(* CODESYS project Structs.export

Project tree, tasks and I/O mapping:
  Structs/
    data type BitByte
    data type udtActuator
    data type udtCamera
    data type udtGeneralBuffer
    data type udtGornModbus
    data type udtTMPBreakingValve
    data type udtVacuumCamera
    DiscreteSignal/
      data type udtDiscreteSignal
      data type udtDiscreteSignalSetting
    Driver/
      data type udtBSDDriver
      data type udtBSDDriverSetting
    FVP/
      data type udtFVP
      data type udtFVPSetting
    GasRegulator/
      data type udtPIDSetting
    Gorn/
      data type udtGorn
      data type udtGornSetting
      Modbus/
        data type GornReadRegister
        data type GornWriteRegister
    HeatfloatSencore/
      data type udtHeatFloatSensore
      data type udtHeatFloatSensoreSetting
    Inficon/
      data type udtInficonGeneralCommand
      data type udtInficonGeneralParameters
      data type udtInficonMaterialParameters
      data type udtInficonProcessMaterialParameters
      data type udtInficonRemoteGeneral
      data type udtInficonRemoteMaterial
      data type udtInficonSensorParameter
      data type udtInficonSourceParameters
      data type udtInficonStatusGeneral
      data type udtInficonStatusMaterial
      data type udtInficonStatusSensor
      InficonType/
        data type InficonFloat
        data type InficonInteger
        data type InficonLong
        data type InficonTime
        BitByte/
          data type InficonInputStatus
          data type InficonLogicstatementStatus
          data type InficonOutputStatus
        Real/
          data type REAL3x1
          data type REAL41
          data type REAL4F31
          data type REAL4x2
          data type REAL5F32
          data type REAL5x3
          data type REAL6F32
    IPS/
      data type udtIPS
      data type udtIPSModbus
      Modbus/
        data type IpsMagnetronReadRegisters
        data type IpsMagnetronWriteRegisters
    Modbus/
      data type sModbusRegister
      data type unRegisterValue
    OWEN/
      data type OwenValue
    OwenAnalogSignal/
      data type udtOwenAnalogSignal
    Pumping/
      VacuumProccessWithSHV/
        data type udtVacuumProccessStatusBitMap
        data type udtVacuumProcess
        data type udtVacuumProcessState
        data type VacuumProccessStatus
        data type VacuumStage
        Devacuum/
          data type DevacuumUnitStage
          data type udtDevacuumUnitProcessSetting
        Revacuum/
          data type RevacuumStage
          data type udtRevacuumProcessSetting
        StartUnitStage/
          data type StartUnitStage
          data type udtStartUnitProcessSetting
        StopUnit/
          data type StopUnitStage
    RRG/
      data type udtRRG
      data type udtRRGSetting
      Modbus/
        data type udtRRGFlagState1
        data type udtRRGFlagState1Flags
        data type udtRRGFlagState2
        data type udtRRGFlagState2Flags
        data type udtRRGModbus
    Shutter/
      data type udtShutter
    TMPDigital/
      data type udtTMPDigital
      data type udtTMPDigitalSetting
    TRM151_Control/
      data type udtTRMHeaterView
      View/
        data type udtTRMChannelView
        data type udtTRMInputView
        data type udtTRMOutput
        Operating/
          data type udtTRMOperatingView
        Regulator/
          data type udtTRMPIDRegualtor
          data type udtTRMRegulatorView
        SetPoints/
          data type udtStepSetPointView
        TechnologProgramm/
          data type udtTRMTechnologOperation
          data type udtTRMTechnologOperationProgram
          data type udtTRMTechnologOperationProgramStep
    TRM151_Protocol/
      data type udtChannel
      data type udtTRM151_01
      Calculator/
        data type udtCalculator
        data type udtCalculatorInput
        data type udtCalculators
      Inputs/
        data type udtInput
        data type udtInputs
      LockAndChangeMode/
        data type udtTRMLockAndChangeMode
      OperationParameters/
        data type udtOperationParameters
        data type udtPowerFeedback
        data type udtSetPointFeedback
      Program/
        data type udtProgram
        data type udtProgramOfTechnolog
        data type udtStep
      Regulators/
        data type udt2PositionRegulator
        data type udtPIDRegulator
        data type udtRegulator
        data type udtRegulators
      SetPoint/
        data type udtProgramSetPoint
        data type udtSetPoints
        data type udtStepSetPoint
      SignalConverter/
        data type udtSignalConverter
        data type udtSignalConverters
    VacuumSensore/
      data type udtAPG100
      data type udtAPG100Setting
      data type udtPressureSensore
      data type udtPressureSensoreSettiing
    Valve/
      data type udtValve
      data type udtValveSetting
*)

// Structs/BitByte
TYPE BitByte :
STRUCT
	b0: BIT;
	b1: BIT;
	b2: BIT;
	b3: BIT;
	b4: BIT;
	b5: BIT;
	b6: BIT;
	b7: BIT;
END_STRUCT
END_TYPE

// Structs/udtActuator
TYPE udtActuator :
	(*Стурктура для Актуатора*)
STRUCT
	xInterlock:				BOOL;// INPUT: Внешняя блокировка
	xOpenInterlock:			BOOL;
	xCloseInterlock:		BOOL;
	xOpenBlocked:			BOOL;
	xCloseBlocked:			BOOL;
	xServiceMode:			BOOL;// COMMAND: Сервисный режим
	xOpenCommand:			BOOL;// COMMAND: Команда на октрытие
	xCloseCommand:			BOOL;// COMMAND: Команда на закрытие
	xOpen:					BOOL;// OUTPUT: Открытие
	xClose:					BOOL;// OUTPUT: Закрытие
END_STRUCT
END_TYPE

// Structs/udtCamera
TYPE udtCamera :
	(*Структура для обработки состояния камеры*)
STRUCT
	xOpened:				BOOL;//INPUT: Камера открыта
	xClosed:				BOOL;//INPUT: Камера закрыта
	xUpPosition:			BOOL;//INPUT: Верхняя позиция
END_STRUCT
END_TYPE

// Structs/udtGeneralBuffer
TYPE udtGeneralBuffer :
STRUCT
	Buffer: POINTER TO BYTE;
	MaxLength: INT;
	Offset: INT;
END_STRUCT
END_TYPE

// Structs/udtGornModbus
TYPE udtGornModbus :
STRUCT
	uiModbusAddress: UINT;//Адрес юнита
	Read:			GornReadRegister;//Список всех регистров на чтение
	Write:			GornWriteRegister;//Список всех регистров на запись
	
END_STRUCT
END_TYPE

// Structs/udtTMPBreakingValve
TYPE udtTMPBreakingValve :
STRUCT
	xAutoMode:			BOOL;//manual/Auto Mode
	xInterlock:			BOOL;
	xManualCommand: 	BOOL;
	xAutoCommand:		BOOL;
	xClosed:			BOOL;
	xOutputCommnad:		BOOL;
END_STRUCT
END_TYPE

// Structs/udtVacuumCamera
(*Структура данных для вакуумнйо камеры*)
TYPE udtVacuumCamera :
STRUCT
	xClosed:								BOOL;	//STATE: Вакуумная камер Открыта/Закрыта
	xCameraIsVaccumed: 						BOOL;	//STATE: Вакуумная система Остановлена/Запущена
	xFVPChecked:							BOOL;	//STATE: Форвакуумный насос прошел проверку
	VacuumCameraProcessStage:				INT;	//STATE: Стадия процесса вакуумной камеры
	
	
	
	rTmpForvacuumingProcessDonePressuresSp: REAL;	//Давление необходимое и достаточное для включения ТМН
	rPressureForVacuumiongProcessComplete:  REAL;	//давление для завершения процесса откачки
	tStopTMPtime:							TIME;  	//Полное время для остановки ТМН
	tOpenBAV3time:							TIME;   //период во времени при полной остановке ТМН когда будет открыьт клапан напуска
	
END_STRUCT
END_TYPE

// Structs/DiscreteSignal/udtDiscreteSignal
TYPE udtDiscreteSignal :
STRUCT
	xSignal:			BOOL;// I/O 

	xValue:				BOOL;// Ready value from/to PLC programms	
END_STRUCT
END_TYPE

// Structs/DiscreteSignal/udtDiscreteSignalSetting
TYPE udtDiscreteSignalSetting :
STRUCT
	xInv:				BOOL;// Инвертирвоанный сигнал
	xSimMode:			BOOL;// Simulation Mode
	xSimValue:			BOOL;// Simulation Value
END_STRUCT
END_TYPE

// Structs/Driver/udtBSDDriver
TYPE udtBSDDriver :
STRUCT
	AutoMode: 			BOOL;	//STATUS
	ServiceMode:		BOOL;	//STATUS
	Blocked:			BOOL;	//STATUS
	Run:				BOOL;	//STATUS
	
	
	
	rSpeedSP:			REAL;	//Setpoint
	
	xAutoCommand:		BOOL;	//COMMAND
	xManualCommand:		BOOL;	//COMMAND
	
	xInterlockSignal: 	BOOL; //Input
	xAlarmSignal:		BOOL; //Input
	
	xStartSignal:		BOOL;
	xCCWSignal:			BOOL;
	rSignal: 			REAL; //OUTPUT: CommandSignal to BSD driver Limit 0-5V
END_STRUCT
END_TYPE

// Structs/Driver/udtBSDDriverSetting
TYPE udtBSDDriverSetting :
STRUCT
	rMinSignalLimit:	REAL;
	rMaxSignalLimit:	REAL;
	rManualSpeedSP:		REAL;
	rAutoSpeedSP:		REAL;
	rMaxSpeed:			INT; //Оборы в минкуту
	xAutoMode:			BOOL;
	xServiceMode:		BOOL;
	xCCWMode:			BOOL;		
END_STRUCT
END_TYPE

// Structs/FVP/udtFVP
TYPE udtFVP :
	(*Структура данных форвакуумного насоса*)
STRUCT
	xPowerOnFeedBack:			BOOL;// INPUT: Обратная связь по питанию
	xInterlock:					BOOL;// INPUT: Внешний сигнал о блокировки
	xManualCommand:				BOOL;// COMMAND: Ручная комманда
	xAutoCommand:				BOOL;// COMMAND: Команда в автоматическом режиме
	xTurnOn:					BOOL;//	STATUS: Насос включен
	xBlocked:					BOOL;// OUTPUT: Сигнал о блокировке 
	xStart:						BOOL;// OUTPUT: Старт/Стоп ФВН
	xPowerOn:					BOOL;// OUTPUT: Состояние питания
END_STRUCT
END_TYPE

// Structs/FVP/udtFVPSetting
TYPE udtFVPSetting :
STRUCT
	xAutoMode:					BOOL;// COMMAND: Автоматическийй/ручной режим
	xServiceMode:				BOOL;// COMMAND: Сервисный режим
	
	xWithOutTurnOn:				BOOL;//Setting: Работа без контактора
END_STRUCT
END_TYPE

// Structs/GasRegulator/udtPIDSetting
TYPE udtPIDSetting :
STRUCT
	rMaunalSP: 	REAL; 	// Расход в литрах РРГ
	rAutoSP:	REAL;	// Необходимое давление.
	rMaxSP:		REAL; 	// Максимальный расход
	rMinSP:		REAL; 	// Минмиальный расход
	iP:			REAL; 	// Пропорциональынй коэффтициент
	tI:			REAL;	// Интегральный коэфф
	rK1RRG:		REAL;	// Коэффитциент РРГ
	rK2RRG:		REAL;
	rK3RRG:		REAL;
	
	xAutoMode:	BOOL;
END_STRUCT
END_TYPE

// Structs/Gorn/udtGorn
TYPE udtGorn :
	(*Стурктура данных для высокотемпературного нагревателя ГОРН
		Верхний уровень управления*)
STRUCT
	
	rSpCurrentFeedback:			REAL;// FEEDBACK: Обратная связь по уставке силы тока
	rSpVoltageFeedback:			REAL;// FEEDBACK: Обратная связь по уставке напряжения
	rFbCurrent:					REAL;// FEEDBACK: Обратная связь по силе тока
	rFbVoltage:					REAL;// FEEDBACK: Обратная связь по напряжению 
	xPowerOnFeedback:			BOOL;// INPUT: Обратная связь по питанию
	xInterlock:					BOOL;// INPUT: Внешняя блокировка
	xRemote:					BOOL;// COMMAND: местынй/дистанционный режимы работы
	xAutoMode:					BOOL;// COMMAND: ручной/автоматический режимы
	xManualCommand:				BOOL;// COMMAND: Команда выкл/вкл в ручном режиме
	xManualPowerCommand:		BOOL;// COMMAND: Команда выкл/вкл питания силовой части в ручном режиме.
	xAutoCommand:				BOOL;// COMMAND: Команда в автоматическом режиме
	xAutoPowerCommand:			BOOL;// COMMAND: Команда питания силовой части в автоматичсеском режиме
	xAcknowledge:				BOOL;// COMMAND: Оператор сбрасывает ошибки
	xBlocked:					BOOL;// STATUS: Заблокирован
	xTurnOn:					BOOL;//	STATUS: В работе
	xError:						BOOL;// STATUS: Общие ошибки
	xInternalError:				BOOL;// OUTPUT: Внутренняя ошибка
	xStabVoltageError:			BOOL;// OUTPUT: Ошибка стабилизации напряжения
	xStabCurrentError:			BOOL;// OUTPUT:	Ошибка стабилизации силы тока
	xPowerError:				BOOL;// OUTPUT: Ошибка силовой части
	xHeatProtect:				BOOL;// OUTPUT: Тепловая защита
	xRemoteStatus:				BOOL;// OUTPUT: Статус удаленной работы
END_STRUCT
END_TYPE

// Structs/Gorn/udtGornSetting
TYPE udtGornSetting :
STRUCT
	rSpCurrent:					REAL;	// SETPOINT: Уставка силы тока
	rSpVoltage:					REAL;	// SETPOINT: Уставка напряжения
	rMaxSpVoltage:				REAL;	// SETTING: Максимальное ограничение на уставку по напряжению
	rMinSpVoltage:				REAL;	// SETTING: Минимальное ограничение на уставку по напряжению
	rMaxSpCurrent:				REAL;	// SETTING: Максимальное ограничение на уставку по силе тока
	rMinSpCurrent:				REAL;	// SETTING: Минимальное ограничение на уставку по силе тока
	iVoltagePointPosition:		INT;	// SETTING: Положение точки в значениях напряжения
	iCurrentPointPosition:		INT;	// SETTING: Положение точки в значениях тока 
END_STRUCT
END_TYPE

// Structs/HeatfloatSencore/udtHeatFloatSensore
TYPE udtHeatFloatSensore :
STRUCT
	rInputTemperature:			REAL;//INPUT: Температура жидкости
	rInputFloat:				REAL;//INPUT: Расход жидкоти в л/ч
	xErrorFloat:				BOOL;//OUTPUT: Ошибка расхода
	xErrorHeat:					BOOL;//OUTPUT: Ошибка температуры
	xTemperatureH:				BOOL;//OUTPUT: Верхний предупредительны сигнал температуры
	xTemperatureHH:				BOOL;//OUTPUT: Верхний аварийный сигнал температуры
	xFloatL:					BOOL;//OUTPUT: Нижний предупредительный сигнал по расходу жидкости
	xFloatLL:					BOOL;//OUTPUT: Нижний авраийный сигнал по расходу жидкости
END_STRUCT
END_TYPE

// Structs/HeatfloatSencore/udtHeatFloatSensoreSetting
TYPE udtHeatFloatSensoreSetting :
STRUCT
	rTemperatureSPH:			REAL;//SETTING: Уставка верхнего предупредительного сигнала температуры
	rTemperatureSPHH:			REAL;//SETTING:	Уставка верхнего аварийного сигнала температуры
	rTemperatureHyst:			REAL;//SETTING: Гистерезис температуры
	rFloatSPL:					REAL;//SETTING: Уставка нижнего предупредительного сигнала расхода жидкости
	rFloatSPLL:					REAL;//SETTING: Уставка нижнего аварийного сигнала расхода жидкости
	rFloatHyst:					REAL;//SETTING: Гистерезис расхода жидкости
END_STRUCT
END_TYPE

// Structs/Inficon/udtInficonGeneralCommand
TYPE udtInficonGeneralCommand :
STRUCT
	Length:		WORD;
	Message:	POINTER TO BYTE;
	Checksum:	BYTE;
	
END_STRUCT
END_TYPE

// Structs/Inficon/udtInficonGeneralParameters
TYPE udtInficonGeneralParameters :
STRUCT
	(*
		Значения являются источниками, толщина которых суммируется
	*)
	ThicknessEq1: 		InficonInteger;
	ThicknessEq2: 		InficonInteger;
	ThicknessEq3: 		InficonInteger;
	Test:				INT; // 0 - Off: 1-On
	TimeCompressed:		INT; // 0-No; 1-Yes
	AdvancedTest:		INT; // 0-Off; 1-On
	AudioFeedback:		INT; // 0-No; 1-Yes
	LCDDimmerTime:		INT; // 0 -AlwaysOn; Minutes till off
	Dateformat:			INT; // 0-mm/dd/yyyy; 1-dd/mm/yyyy
	USBDatalogFormat:	INT; // 0-Log off; 1-page; 2-Command
	DatalogXtalInfo:	INT; // 0-No; 1-Yes
	(*Обновление изменит все графики материалов на выбор шкалы графиков.*)
	GraphScale:			INT; // 0-Power; 1- 10A/s 2- 20A/s
	GraphScanRate:		INT; // 0-Auto; 1-Slow; 2-Medium; 3-Fast
	RS232BaudRate:		INT; // 0-9600; 1-19200; 2-38400; 3-57600; 4-115200
	RS232Protocol:		INT; // 0-standart; 1-DlogPage; 1-Dlog Command
	DAC1Scale:			REAL3x1;
	DAC2Scale:			REAL3x1;
	DAC3Scale:			REAL3x1;
	DAC4Scale:			REAL3x1;
	DAC5Scale:			REAL3x1;
	DAC6Scale:			REAL3x1;
	DAC7Scale:			REAL3x1;
	DAC8Scale:			REAL3x1;
	DAC9Scale:			REAL3x1;
	DAC10Scale:			REAL3x1;
	DAC11Scale:			REAL3x1;
	DAC12Scale:			REAL3x1;
	DAC1Polarity:		INT; // 0 -Negative 1-Positive
	DAC2Polarity:		INT; // 0 -Negative 1-Positive
	DAC3Polarity:		INT; // 0 -Negative 1-Positive
	DAC4Polarity:		INT; // 0 -Negative 1-Positive
	DAC5Polarity:		INT; // 0 -Negative 1-Positive
	DAC6Polarity:		INT; // 0 -Negative 1-Positive
	DAC7Polarity:		INT; // 0 -Negative 1-Positive
	DAC8Polarity:		INT; // 0 -Negative 1-Positive
	DAC9Polarity:		INT; // 0 -Negative 1-Positive
	DAC10Polarity:		INT; // 0 -Negative 1-Positive
	DAC11Polarity:		INT; // 0 -Negative 1-Positive
	DAC12Polarity:		INT; // 0 -Negative 1-Positive
	(* 0 -Power; 1 - 0.1A/s; 2 - 0.5A/s; 3 - 1A/s; 4 - 2A/s;
 	5 - 3A/s; 6 - 5 A/s; 7 - 10A/s: 8 - 20A/s; 9 - 50A/s*)
	Channel1GraphScale:	INT; 
	Channel2GraphScale:	INT; 
	Channel3GraphScale:	INT; 
	Channel4GraphScale:	INT; 
	Channel5GraphScale:	INT; 
	Channel6GraphScale:	INT; 
END_STRUCT
END_TYPE

// Structs/Inficon/udtInficonMaterialParameters
TYPE udtInficonMaterialParameters :
STRUCT
	Density:			REAL5x3;
	ZRatio:				REAL5x3;
	MasterTooling:		REAL41;
	ControlLoop:		INT;//0-NonPID; 1-PI; 2-PID
	ProcessGain:		REAL5F32;
	TimeConstant:		REAL6F32; // Seconds. Gray font if Control Loop - Non PID
	DeadTime:			REAL6F32; // Seconds. Gray font if Control Loop - Non PID
	MaximumPower: 		REAL4x2;
	MinimumPower:		REAL4x2;
	MaxPowerEncode:		INT; // 0 - Continue; 1 - Post-Dep; 2-Stop All; 3 - Stop Matl
	PreCondRiseTime: 	InficonTime; // Maximum time 5999 seconds, Displayed as 99:59
	PreCondSoakTime:	InficonTime;
	SoakPower1:			REAL4x2;
	RiseTime1:			InficonTime;
	SoakTime1:			InficonTime;
	SoakPower2:			REAL4x2;
	RiseTime2:			InficonTime;
	SoakTime2:			InficonTime;
	AutoSoak2:			INT;	//0-No; 1-Yes;
	DepAfterPreDep:		INT;	//0-No; 1-Yes
	DelayOption:		INT;	//0-None; 1-Shutter; 2-Control: 3-Both
	ControlDelayTime:	InficonTime;
	ShutterDelayAccur:	InficonInteger;// %l Default -5;
	FeedPower:			REAL4x2;
	FeedRampTime:		InficonTime;
	FeedTime:			InficonTime;
	IdlePower:			REAL4x2;
	IdleRampTime:		Inficontime;
	Rate:				REAL4F31; // A/s
	TimeLimit:			InficonTime;
	RateFilterTime:		INT; // 0 - 0.1; 1 - 0.4; 2 - 1.0; 3 - 4.0; 4 - 10.0; 5- 20.0; 6 - 30.0;
	TimePowerAvgTime:	InficonInteger; //Minutes
	IonAssistDeposit:	INT; //0-No; 1-YES;
	OnFinalthickness:	INT; //0-Continue; 1-Post-Dep; 2-NonDepCont
	Ramp1Rate:			REAL4F31;
	StartRamp1:			REAL4F31;
	Ramp1Time:			InficonTime;
	Ramp2Rate:			REAL4F31;
	StartRamp2:			REAL4F31;
	Ramp2Time:			InficonTime;
	RateWatcherOption:	INT; //	0- No; 1-Yes;
	RateWatcherTime:	InficonTime;
	RateWatcherAccurace:InficonInteger;//%	
	FailureAction:		INT;// Default -3; 1-PostDp; 2-StopAll; 3-StopMatl; 4-TimePW
	CrystalTwoTooling:	REAL41;
	XtalPositionFirst:	InficonInteger; // 0-12
	XtalPositionLast:	InficonInteger; // 0-12
	QualityPercent:		InficonInteger; //% 0 -99
	QualityCounts:		InficonInteger;
	StabilitySingle:	InficonInteger; // 0-9999
	StabilityTotal:		InficonInteger;	// 0-9999
	RecorderOutput:		InficonInteger;
	RecorderFunction:	INT; //0-FilteredRate; 1-Thick; 2-RateDev; 3-Power
	RecorderRange:		InficonInteger;
	
END_STRUCT
END_TYPE

// Structs/Inficon/udtInficonProcessMaterialParameters
TYPE udtInficonProcessMaterialParameters :
STRUCT
	FinalThick:				REAL5F32;//kA
	ThickLimit:				REAL5F32;
	Crucible:				InficonInteger;
END_STRUCT
END_TYPE

// Structs/Inficon/udtInficonRemoteGeneral
TYPE udtInficonRemoteGeneral :
STRUCT
	StopAll:						BOOL;
	ResetAll:						BOOL;
	RemoteLockOn:					BOOL;
	RemoteLockOff:					BOOL;
	SetLogicStatement:				BYTE;
	ClearLogicStatement:			BYTE;
	CrystalFailInhibitOn:			BYTE;
	CrystalFailInhibitOff:			BYTE;
	SetDate:						ARRAY[0..2] OF InficonInteger;
	SetTime:						ARRAY[0..2] OF InficonInteger;
	ZeroCounter:					BYTE;
	ZeroTimer:						BYTE;
	StartTimer:						BYTE;
	ClockHoldOn:					BYTE;
	ClockHoldOff:					BYTE;
	UserMessageOn:					BYTE;
	UserMessageOff:					BYTE;
	SoakHold1On:					BYTE;
	SoakHold1Off:					BYTE;
	SoakHold2On:					BYTE;
	SoakHold2Off:					BYTE;
	SwitchSensor:					ARRAY[0..1] OF BYTE;
	ClearFailedCrystalsX:			BYTE;
	RotateHeadX:					BYTE;
	DefaultAllParameters:			BOOL;
	SoakHoldPreConOn:				BYTE;
	SoakHoldPrecomOff:				BYTE;
	StartInhibitOn:					BOOL;
	StartIngibitOff:				BOOL;
	RateWatcherSamplingInhibitOn:	BYTE;
	RateWatcherSamplingInhibitOff:	BYTE;
	WatcherSamplingInitiateOn:		BYTE;
	WatcherSamplingInitiateOff:		BYTE;
	ClearQAndSCountsForSensore:		BYTE;
	NameMaterial:					ARRAY[0..1]OF BYTE;
END_STRUCT
END_TYPE

// Structs/Inficon/udtInficonRemoteMaterial
TYPE udtInficonRemoteMaterial :
STRUCT
	StopMaterial:			BOOL;
	ZeroThickness:			BOOL;
	StartDeposit:			BOOL;
	GoToNonDepositControl:	BOOL;
	GoToPostDeposit:		BOOL;
	ContinueDeposit:		BOOL;
	GoToManual:				BOOL;
	SetPowerlevel:			InficonFloat;
	OpenSourceShutter:		BOOL;
	CloseSourceShutter:		BOOL;
	SetAverageRate:			InficonFloat;
	Start:					BOOL;
	ResetMaterial:			BOOL;
END_STRUCT
END_TYPE

// Structs/Inficon/udtInficonSensorParameter
TYPE udtInficonSensorParameter :
STRUCT
	ShutterOut:			InficonInteger;
	SensorType:			INT;// 0-single; 1-XtalTwo; 2-XtalSix; 3-Xtal12; 4-Generic
	SwitchOut:			InficonInteger;
	AutoZ:				INT;// 0 - No; 1-Yes
	(*Visible only sensor type = 4*)
	NumberOfPosition:	InficonInteger;
	NumberOfPulse:		InficonInteger;
	PulseOn:			REAL3x1; //Second
	PulseOff:			REAL3x1; //Second
	//------------------------------
	RecorderOutput:		InficonInteger;
	RecorderFunction:	INT; //0 - Unifiltered Rate; 1- thick; 2- RateDev
	RecorderRange:		InficonInteger;
	
END_STRUCT
END_TYPE

// Structs/Inficon/udtInficonSourceParameters
TYPE udtInficonSourceParameters :
STRUCT
	DACOutput:			InficonInteger;
	ShutterOutput:		InficonInteger;
	NumberOfCrucibles:	INT; // Число тигелей 0-1; 1-4; 2-8; 3-16; 4-32; 5-64 
	CrucibleOutput:		InficonInteger;
	TurretFeedback:		INT; // 0 -No; 1-Yes
	TurretInput:		InficonInteger;
	TurretDelay:		InficonInteger; // Seconds
	
END_STRUCT
END_TYPE

// Structs/Inficon/udtInficonStatusGeneral
TYPE udtInficonStatusGeneral :
STRUCT
	OutputStatus: 				InficonOutputStatus; //Responce - 5 bytes. Каждый бит репрезентует OUTPUT
	InputStatus:				InficonInputStatus; //Responce - 4 bytes
	LogicStatementStatus:		InficonLogicstatementStatus;//Responce - 13 byte
	StatusMessage:				ARRAY [0..7] OF BYTE; //Responce - 8 bytes
	StatusMessageDesignators:	ARRAY [0..12] OF BYTE;
	TrancientMessages:			BYTE; // Responce - 1 bytes
	SensorStatus:				ARRAY [0..5] OF BYTE;
	TimerStatus:				BYTE;
	TimerValue:					InficonInteger;
	CounterValue:				InficonInteger;
	ThicknessSum:				ARRAY [0..2] OF REAL3x1;
	GetDate:					ARRAY [0..2] OF InficonInteger;
	GetTime:					ARRAY [0..2] OF InficonInteger;
	SystemConfuguration:		ARRAY[0..1] OF BYTE;
END_STRUCT
END_TYPE

// Structs/Inficon/udtInficonStatusMaterial
TYPE udtInficonStatusMaterial :
STRUCT
	FilteredRate:			ARRAY [0..5] OF InficonFloat; // A/s
	DisplayRate:			ARRAY [0..5] OF InficonFloat; // A/s
	SourcePowerOutput:		ARRAY [0..5] OF InficonFloat; // %;
	Thickness:				ARRAY [0..5] OF InficonFloat; // kA
	State:					ARRAY [0..5] OF BYTE;
	StateTime:				ARRAY [0..5] OF InficonInteger;
	ActiveSensors:			ARRAY [0..5] OF BYTE;
	PowerSourceNumber:		ARRAY [0..5] OF BYTE;
	AccumulatedLayerTime:	ARRAY [0..5] OF InficonInteger;
	DepositAverageRate:		ARRAY [0..5] OF InficonFloat; // kA
	DepositAveragePower:	ARRAY [0..5] OF InficonFloat; // %
	RawRate:				ARRAY [0..5] OF InficonFloat; // kA
	OneMinuteAvgForRatePwr:	ARRAY [0..11] OF InficonFloat;;
	RateDeviation:			BYTE:=16#0E;
	StateBeforeStop:		ARRAY [0..5] OF BYTE;
	DataLog:				BYTE:=16#10;
	DataLogwithXtalHistory:	BYTE:=16#11;
	CauseOfStop:			ARRAY [0..5] OF BYTE;	
END_STRUCT
END_TYPE

// Structs/Inficon/udtInficonStatusSensor
TYPE udtInficonStatusSensor :
STRUCT
	CrystalLife:		ARRAY [0..5] OF BYTE;
	CrystalsRemaning:	ARRAY [0..5] OF BYTE;
	CrystalPosition:	ARRAY [0..5] OF BYTE;
	SensorStatus:		ARRAY [0..5] OF BYTE;
	FundamentalFreq:	ARRAY [0..5] OF InficonLong; // KtoHz=0.000873114913702011
	FundamentalActivity:ARRAY [0..5] OF InficonInteger;
	CurrentZRation:		ARRAY [0..5] OF InficonFloat;
	AnharmonicFreq:		ARRAY [0..5] OF InficonLong;
	AnharmonicActivity:	ARRAY [0..5] OF InficonInteger;
	NewCrtystaFreq:		ARRAY [0..11] OF InficonLong;
	LCQValue:			ARRAY [0..5] OF InficonFloat;
	SensorThickness:	ARRAY [0..5] OF InficonFloat;
END_STRUCT
END_TYPE

// Structs/IPS/udtIPS
TYPE udtIPS :
STRUCT
	xInterlock: 					BOOL;//Input: Внешняя блокировка
	xPowerOnFeedback:				BOOL;//Input: Обратная связь по питанию.
	rCurrentFeedback:				REAL;//Input: ОБратная связь по напряжению
	rVoltageFeedback:				REAL;//Input: Обратная связь по напряяжени.
	rPowerFeedback:					REAL;//Input: Обратная связь по мощности
	xTurnOn:						BOOL;//Input: Включен
	xError:							BOOL;//Input: ОШИБКА
	sStatus:						STRING;//Input: СТАТУС
	
	xDeviceSwitchOn:				BOOL;//STATUS: Блок в целом включен 0-бит
	xSmoothIncreseOutParametr:		BOOL;//STATUS: Режим плавного увеоичения выходного параметра с заданной скоростью 2-БИТ
	xSmoothDecreaseOutParametr:		BOOL;//STATUS: Режим плавного уменьшения выходного параметра с заданной скоростью 3-БИТ
	xInputConverterSwitchOn:		BOOL;//STATUS: Хотя бы один выходной преобразователь включен 4-БИТ	
	xInputPowerOutOfLimit:			BOOL;//STATUS: Входная сеть вне допустимого диапозона
	xCriticalTemeratureWarning:		BOOL;//STATUS: Температура блока близка к критической
	xOverload:						BOOL;//STATUS: перегрзука блока Питания
	xOutPowerSitchingOn:			BOOL;//STATUS: Идет включение выходного напряжения
	xOutPowerSwitchingOff:			BOOL;//STATUS: Идет выключение выходного напряжения
	xCrititicalCurrentPulseWarning:	BOOL;//STATUS: Пульсация тока в нагрузке близка к критической
	xBuzzerOn:						BOOL;//STATUS: Включение звукового сигнала
	xDisplayConnect:				BOOL;//STATUS: Связь с дисплеем 13
	xADCEnable:						BOOL;//STATUS: АЦП присутствует, блок питаняи в норме 15
	xBlocked:						BOOL;//STATUS: Блокировка

	
	xAutoMode:						BOOL;//SETTING: Автоматичсекий режим
	xService:						BOOL;//SETTING: Сервисный режим
	xRemote:						BOOL;//SETTING: Удаленный режим
	rPowerSp:						REAL;//SETTING: Уставка по мощности
	rCurrentSP:						REAL;//SETTING:	Уставка по току
	rVoltageSP:						REAL;//SETTING: Уствка по напряжению
	rPowerSpMin:					REAL;//SETTING: Минимальное значение уставки по мощности
	rPowerSpMax:					REAL;//SETTING: максимальное значение уставки по мощности
	rCurrentSpMin:					REAL;//SETTING: Минимальное значение устваки по току
	rCurrentSpMax:					REAL;//SETTING:	Максимальное значение уствки по току
	rVoltageSpMin:					REAL;//SETTING: Минимальное значение уставки по напряжению
	rVoltageSpMax:					REAL;//SETTING:	Максимальное значение уставки по напряжению
	
	xManualStartCommand:			BOOL;//COMMAND:	Ручная комманда
	xManualStopCommand:				BOOL;//COMMAND:	Ручная комманда
	xAutoStartCommand:				BOOL;//COMMAND:	Автоматическая команад
	xAutoStopCommand:				BOOL;//COMMAND:	Автоматическая команад
	xErrorReset:					BOOL;//COMMAND: Сброс ошибок
	
	xStart:							BOOL;//OUTPUT:	Команда на старт 
	xStop:							BOOL;//OUTPUT: Команда на стоg
	xReset:							BOOL;//OUTPUT: Сброс ошибок
	
	
	
	
END_STRUCT
END_TYPE

// Structs/IPS/udtIPSModbus
TYPE udtIPSModbus :
STRUCT
	uiAddress:		UINT;// АДРЕС
	Read:			IpsMagnetronReadRegisters;
	Write:			IpsMagnetronWriteRegisters;
END_STRUCT
END_TYPE

// Structs/Modbus/sModbusRegister
{info "@TODO дописать структуру, исходя из логики приема передачи"}
TYPE sModbusRegister :
STRUCT
	iRegister:	INT; //Адрес регистра/Смещение/Offset
	sValue:		unRegisterValue; //Значение в регистре
END_STRUCT
END_TYPE

// Structs/Modbus/unRegisterValue
TYPE unRegisterValue :
	(*Регистр состояни истояника питания и регистр управления источником питаня для Рабочих параметров ГОРН*)
UNION
	COIL_VALUE: 	ARRAY[0..15] OF BOOL; 
	WORD_VALUE: 	WORD;
	INT_VALUE:		DINT;
END_UNION
END_TYPE

// Structs/OWEN/OwenValue
TYPE OwenValue :
STRUCT
	ID:											WORD:=16#FF;
	ParameterName:								STRING; //имя параметра
	ValueType:									OWEN_TYPE;//Тип данных
	IntValue:									DINT;
	FloatValue:									REAL;
	OtherValue:									ARRAY[0..15] OF BYTE;
END_STRUCT
END_TYPE

// Structs/OwenAnalogSignal/udtOwenAnalogSignal
(*Стурктура для аналоговых входных сигналов Owen MK210-*)
TYPE udtOwenAnalogSignal :
STRUCT
	rSignal: 			REAL;// Signal from/to PLC 
	rSimValue:			REAL;// Simulation Value
	rValue:				REAL;//	Value from/to PLC program
	xSimMode:			BOOL;// Enable/Disable Simulation Mode;
  
END_STRUCT
END_TYPE

// Structs/RRG/udtRRG
TYPE udtRRG :
STRUCT
	rManualValueSP: 	REAL; // ручной расход в литрах
	rAutoValueSP: 		REAL; //автмоатический расход в процентах
	rValueSP:			REAL; //
	
	
	rSetPointFeedback:	REAL;
	rValueFeedback:		REAL;
	
	xError:					BOOL;
	
	
	xDigitalInputFeedback: 	BOOL;//
	xValveOpenFeedback: 	BOOL;
	xValveCloseFeedback: 	BOOL;
	xValveRegModeFeedback:	BOOL;
	xRepaireModeFeedback:	BOOL;
	xRRGModeFeedback:		BOOL;//0-RRG; 1-RDG
	
	(*Flag State 2*)
	xLowGasFlow:			BOOL;
	xValveMode:				BOOL;//0- Reg: 1-Discrete
	xRegMode:				BOOL;//0-RRG$ 1-RDG
	xOnlyRDG:				BOOL;
	xOnlyRRG:				BOOL;
	xValveOpenState: 		BOOL;
	xValveCloseState: 		BOOL;
	xValveRegModeState:		BOOL;
	
END_STRUCT
END_TYPE

// Structs/RRG/udtRRGSetting
TYPE udtRRGSetting :
STRUCT
	rMinValue: REAL; //Минимальное значение расхода
	rMaxValue: REAL; //максимальное значение расхода
	xAutoMode: BOOL; //0 -Manual Mode; 1-Auto mode
	xService:  BOOL;
	
	
	
	
	
	xDigitalInputSP: 	BOOL;// 0 - analog: 1 - Digital
	xValveOpenSP: 		BOOL;
	xValveCloseSP: 		BOOL;
	xValveRegModeSP:	BOOL;
	xRepaireModeSP:		BOOL;
	xRRGModeSP:			BOOL;//0-RRG; 1-RDG
END_STRUCT
END_TYPE

// Structs/Shutter/udtShutter
TYPE udtShutter :
STRUCT
	AutoMode: 				BOOL;
	AutoCommand:			BOOL;
	ManualCommand:			BOOL;
	FinallyCommand:			BOOL;
	Interlock:				BOOL;
	ShutterOpened: 			BOOL;
	OpenCommand:			BOOL;
	CloseCommand:			BOOL;
END_STRUCT
END_TYPE

// Structs/TMPDigital/udtTMPDigital
TYPE udtTMPDigital :
	(*Структура ТМН для управления через Remote I/O*)
STRUCT
	xPowerOnFeedBack:			BOOL;// INPUT: Обратная связь по питанию
	xInterlock:					BOOL;// INPUT: Внешний сигнал о блокировки
	xNormalOperation:			BOOL;// INPUT: Сигнал о том что ТМН запущен
	xWarning:					BOOL;// INPUT: Сигнал о предупреждении с ТМН
	xError:						BOOL;// INPUT: Сигшнал об ошибке с ТМН
	xManualCommand:				BOOL;// COMMAND: Ручная комманда
	xAutoCommand:				BOOL;// COMMAND: Команда в автоматическом режиме
	xAutoMode:					BOOL;// COMMAND: Автоматическийй/ручной режим
	xServiceMode:				BOOL;// COMMAND: Сервисный режим
	xAckError:					BOOL;// COMMAND: Сброс сообщения об ошибки ТМН
	
	rMinimalAccessPressure:		REAL;// SETTING: Минимальное давление для заупска ТМН
	
	xPumpNotOperating:			BOOL;
	xPumpIsDecelerating:		BOOL;
	xJustAfterStop:				BOOL;
	xJustAfterStart:			BOOL;
	xPumpIsAccelerating:		BOOL;
	xPumpNormalOperatingMode:	BOOL;
	errPumpStandstill:			BOOL;
	errPumpIsDecelerating:		BOOL;
	errJustOccured:				BOOL;
	
	
	xMore90hzRotate:			BOOL;
	xPumpRotate:				BOOL;
	
	xBreakingValve:				BOOL;// OUTPUT: Сигнал об открытии тормозного клапана
	xBlocked:					BOOL;// OUTPUT: Сигнал о блокировке 
	xStart:						BOOL;// OUTPUT: Старт/Стоп ТМП
END_STRUCT
END_TYPE

// Structs/TMPDigital/udtTMPDigitalSetting
TYPE udtTMPDigitalSetting :
STRUCT
	rMinimalCameraPressure:		REAL;// SETTING: Минимальное давление для заупска ТМН
	rMinimalForvaccumLinePressure: REAl;// SETTING: Минимальное давление в форвакуумной линии для запуска ТМН.
	
END_STRUCT
END_TYPE

// Structs/TRM151_Control/udtTRMHeaterView
TYPE udtTRMHeaterView :
STRUCT
	xPowerOn:					BOOL;//INPUT: Автомат включен
	xInterlock:					BOOL;//INPUT: Внешняя блокирвока
	
	
	

	
	
	xStartCommand:				TRMStartSignal;//COMMAND: Старт работы
	xSaveChannel:				BOOL;//COMMAND: Сохранение настроек канала
	xSaveInput:					BOOL;//COMMAND: Сохранениен настроек ввода
	xSaveRegulator:				BOOL;//COMMAND: Cохранение настроек Регулятора
	xSaveOutput:				BOOL;//COMMAND: Сохранение настроек Выхода
	xSaveStartProgramAndStep:	BOOL;//COMMAND:	Сохранение программы и шага xSaveOperating
	xAutoMode:					BOOL;//COMMAND:	Ручной/Авто режим
	xAutoStart:					BOOL;//COMMAND: Команда в автоматическом режиме
	xAutoStop:					BOOL;
	xManualStart:				BOOL;//COMMAND:	Команда в ручном режиме
	xManualStop:				BOOL;
	xRemoreLocalMode:			BOOL;//COMMAND: Местный/Дистанционный режим
	xServiceMode:				BOOL;//COMMAND: Севрисный режим
	Status:						TRMObjectState;//STATUS: Статус системы
	xBlocked:					BOOL;//STATUS: Заблокирвоан
	
	xRemoteMode:				BOOL;//OUTPUT: Диcтанционный режим работы					 
END_STRUCT
END_TYPE

// Structs/TRM151_Protocol/udtChannel
TYPE udtChannel :
STRUCT
	ChannelNumber:	INT;
	ChannelLoadingIndication: 	OwenValue:=(ParameterName:='S.SAU', ValueType:=OWEN_TYPE.INTEGER); //Семафор загруженности канала (0..255)
	Regulator: 					OwenValue:=(ParameterName:='rEGL', 	ValueType:=OWEN_TYPE.INTEGER);//Регултятор в канале
	Inspector:					OwenValue:=(ParameterName:='insP', 	ValueType:=OWEN_TYPE.INTEGER);//Инспектор в канале
	GroupAttruibute: 			OwenValue:=(ParameterName:='Ch', 	ValueType:=OWEN_TYPE.INTEGER);//Групповой Атрибут канала; 0-не редактируемый. Заводской; 1-Редактируемый,Заводской; 2-Не редактируемый, пользоватлеьский; 3- Редактируемый пользовательский
	
END_STRUCT
END_TYPE

// Structs/TRM151_Protocol/udtTRM151_01
TYPE udtTRM151_01 :
STRUCT
	Channel: 			ARRAY[0..1] OF udtChannel;
	Inputs: 			udtInputs;
	Programs: 			udtProgramOfTechnolog;
	Regulators:			udtRegulators;
	ProgramSetPoint:	udtProgramSetPoint;
	SignalConverters:	udtSignalConverters;
	
	LockAndChangeMode:	udtTRMLockAndChangeMode;
	
END_STRUCT
END_TYPE

// Structs/VacuumSensore/udtAPG100
(*Пользовательский тип данных для форвакуумного датчика*)
TYPE udtAPG100 EXTENDS udtPressureSensore :
STRUCT

	xAtmosphere:		BOOL;//OUTPUT: Атмосфера
	xForVacuum:			BOOL;//OUTPUT: Форвакуум
END_STRUCT
END_TYPE

// Structs/VacuumSensore/udtAPG100Setting
TYPE udtAPG100Setting EXTENDS udtPressureSensoreSettiing :
STRUCT
	rForVacuumSp:		REAL;//SETTING: Уставка давления, ниже которой наступает форвакуум
	rForVacuumHist:		REAL;//SETTING: Гистерезис для показания форвакуума
END_STRUCT
END_TYPE

// Structs/VacuumSensore/udtPressureSensore
(*Струкута для датчика давления WRG и APG*)

TYPE udtPressureSensore :
STRUCT 
	rVolatgeSignal:		REAL;			// INPUT: VOLTAGE SIGNAL

	rPressure:			REAL;			// OUTPUT: VALUE
	sUnit:				STRING;			// OUTPUT: 'mBar', 'Pa', 'Torr'		
	xError:				BOOL;			// OUTPUT: Ошибка модуля
	
END_STRUCT
END_TYPE

// Structs/VacuumSensore/udtPressureSensoreSettiing
(*Настройки для датчиков давления WRG b APG*)
TYPE udtPressureSensoreSettiing :
STRUCT
	rVolageDeathband:	REAL;			// SETTING: Мертвая зона показаний
	rSimValue:			REAL;			// SETTING: Значение давления в режиме симуляции
	enumPressureUnit:	INT;	// SETTING: Какое давление используем
	rKVoltage:			REAL:=1.5;			// SETTING: коэффициент на который умножается вольтовый сигнал в степени
	rKMBar: 			REAL:=12.0;			// SETTING: Коэффициент, который вычитается в степени для мБар
	rKPa:				REAL:=10.0;			// для Па
	rKTorr: 			REAL:=12.125;			// для Torr
	xSimMode:			BOOL;			// SETTING: Режим симуляции	
END_STRUCT
END_TYPE

// Structs/Valve/udtValve
TYPE udtValve :
	(*Струкутура для Клапанов*)
STRUCT
	wInterlockStatus:	WORD;// STATUS: Стаутс блокировки статуса
	xOpened:			BOOL;// INPUT: Сигнал с концевика об открытии клапана
	xClosed:			BOOL;// INPUT: Сигнал о закрытии клапана
	xInterlock:			BOOL;// INPUT: Внешняя блокировка
	xManualCommand:		BOOL;// COMMAND: Команда в ручном режиме
	xAutoCommand:		BOOL;// COMMAND: Команада в автоматическом режиме
	
	
	xError:				BOOL;// OUTPUT: Ошибка клапана
	xBlocked:			BOOL;// OUTPUT: Сигнал о блокировке
	xOpen:				BOOL;// OUTPUT: Сигнал на открытие
	xClose:				BOOL;// OUTPUT: Сигнал на закрытие
	
END_STRUCT
END_TYPE

// Structs/Valve/udtValveSetting
TYPE udtValveSetting :
STRUCT
	xAutoMode:					BOOL;// COMMAND: ручной/Автоматический режимы
	xServiceMode:				BOOL;// COMMAND: Сервисный режим
	xOnlycCloseEnderMode:		BOOL;// SETTING: Режим работы с одним концевиком
	tGripTime:					TIME;// INPUT: Время перед блокировкой
END_STRUCT
END_TYPE

// Structs/Gorn/Modbus/GornReadRegister
TYPE GornReadRegister :
	(*Регистры для чтения ГОРН*)
STRUCT
	strPowerSupplyStatusRegister: 		sModbusRegister;//Регистр состояния блока питания
	strPowerSupplyControlRegister:		sModbusRegister;//Регистар управления блока питания
	strSpCurrent:						sModbusRegister;//Регистр уставки силы тока
	strSpVoltage:						sModbusRegister;//Регистр уставки напряжения
	strFbCurrent:						sModbusRegister;//Регистр измеренного тока
	strFbVolatge:						sModbusRegister;//Регистр ищмеренного напряжения
END_STRUCT
END_TYPE

// Structs/Gorn/Modbus/GornWriteRegister
TYPE GornWriteRegister :
STRUCT
	strPowerSupplyControlRegister:		sModbusRegister;//Регистар управления блока питания
	strSpCurrent:						sModbusRegister;//Регистр уставки силы тока
	strSpVoltage:						sModbusRegister;//Регистр уставки напряжения
END_STRUCT
END_TYPE

// Structs/Inficon/InficonType/InficonFloat
TYPE InficonFloat : DWORD; END_TYPE

// Structs/Inficon/InficonType/InficonInteger
TYPE InficonInteger : DWORD; END_TYPE

// Structs/Inficon/InficonType/InficonLong
TYPE InficonLong : ARRAY[0..7] OF BYTE; END_TYPE

// Structs/Inficon/InficonType/InficonTime
TYPE InficonTime :
STRUCT
END_STRUCT
END_TYPE

// Structs/IPS/Modbus/IpsMagnetronReadRegisters
TYPE IpsMagnetronReadRegisters :
STRUCT
	strCommandAndStatus:		sModbusRegister;//регистр комманд и состояний. 
 	strDevicerStatus:			sModbusRegister;//Состояние устройства
	strLightDiodState:			sModbusRegister;//Состояние светодиодов индикации на передней панели
	srrWorktimer:				sModbusRegister;//Время для работы
	strDeviceCode:				sModbusRegister;//Код устрйоства
	strVersion:					sModbusRegister;//версия программного обеспечения
	strCurrentSP:				sModbusRegister;//Уставка тока
	strVoltageSP:				sModbusRegister;//Уставка напряжения
	strPowerSP:					sModbusRegister;//Уставка мощности
	strCurrenFeedback:			sModbusRegister;//Выходной ток
	strVoltageFeedBack:			sModbusRegister;//Выходное напряжение
	strPowerFeedback:			sModbusRegister;//Выходная мощность
	strEdgeFrontSpeed:			sModbusRegister;//Скорость фронта
	sreEdgeFallSpee:			sModbusRegister;//Скорость спада
	strDealyChannel:			sModbusRegister;//Канал задержки
	strWorkedTime:				sModbusRegister;//Время работы
	strStateFlag:				sModbusRegister;//Флаги состояний
	strNetworkFlag:				sModbusRegister;//Флаг сети. Служебная информация
	strLanguageMenu:			sModbusRegister;//Язык меню
	strInterfaceType:			sModbusRegister;//Тип Интерфейса
	strNetworkAddress:			sModbusRegister;//Сетевой адрес
	strBauldrate:				sModbusRegister;//Скорость связи
	strParity:					sModbusRegister;//Четность		
	strMode:					sModbusRegister;//Режим работы
	strSparkVoltage:			sModbusRegister;//Напряжение дуги для срабатывания системы дугогашения
	strSparkCounter:			sModbusRegister;//счетчик дуг				
	strShutdownDelay:			sModbusRegister;//Задержка отключения
	strTemperature:				sModbusRegister;//температура наиболее нагретого радиатора
	strIcoeff:					sModbusRegister;//pId
	strPcoeff:					sModbusRegister;//Pid
END_STRUCT
END_TYPE

// Structs/IPS/Modbus/IpsMagnetronWriteRegisters
TYPE IpsMagnetronWriteRegisters :
STRUCT
	strCommandAndStatus:		sModbusRegister;// регистр команд и состояний
	
	
	strWorkTime:				sModbusRegister;//время работы
	
	
	strCurrentSP:				sModbusRegister;
	strVoltageSP:				sModbusRegister;
	strPowerSP:					sModbusRegister;
	
	
	
	strEdgeFrontSpeed:			sModbusRegister;//Скорость фронта
	strEdgeFallSpeed:			sModbusRegister;//Скорость спада
	strDelayChannel:			sModbusRegister;//Канал задержки
	
	
	
	strLanguageMenu:			sModbusRegister;
	strInterfaceType:			sModbusRegister;
	strNetworkAddress:			sModbusRegister;
	strBauldrate:				sModbusRegister;
	strParity:					sModbusRegister;
	strkMode:					sModbusRegister;
	strSparkVoltage:			sModbusRegister;
	
	strShutdownDelay:			sModbusRegister;
	
	strIcoeff:					sModbusRegister;
	strPcoeff:					sModbusRegister;
END_STRUCT
END_TYPE

// Structs/Pumping/VacuumProccessWithSHV/udtVacuumProccessStatusBitMap
TYPE udtVacuumProccessStatusBitMap :
STRUCT
	BAV1NotAutoMode: 		BIT;
	BAV2NotAutoMode: 		BIT;
	BAV3NotAutoMode: 		BIT;
	SHVNotAutoMode: 		BIT;
	FVPNotAutoMode: 		BIT;
	TMPNotAutoMode: 		BIT;
	FVPNotPowerOn:			BIT;
	TMPNotPowerOn:			BIT;
	StartStatusProcessError:BIT;	
	
END_STRUCT
END_TYPE

// Structs/Pumping/VacuumProccessWithSHV/udtVacuumProcess
TYPE udtVacuumProcess :
STRUCT
	
	Stage:					INT;
	Status:					VacuumProccessStatus;
	
	UnitTurnOn:				BOOL; //STATUS: Вакуумное оборудование установки включено
	UnitTurnOff:			BOOL; //STATUS: Вакуумное оборудование установки выключено
	VacuumedUnit:			BOOL; //STAUTS: Установка под вакуумом
	DevacuumedUnit:			BOOL; //STATUS: Установка под атмосферой 
	
	
	xStartUnit:				BOOL; //COMMAND: Включение установки
	xStartRevacuumProccess: BOOL; //COMMAND: Старт алгоритма откачки
	xStartDevacuumProcess: 	BOOL; //COMMAND: Старт алгоритма напуска
	xStopUnit:				BOOL; //COMMAND: Выключение установки
	ResetError:				BOOL; //COMMAND: Сброс ошибок
END_STRUCT
END_TYPE

// Structs/Pumping/VacuumProccessWithSHV/udtVacuumProcessState
TYPE udtVacuumProcessState :
STRUCT
	UnitTurnOn:				BOOL; //STATUS: Вакуумное оборудование установки включено
	UnitTurnOff:			BOOL; //STATUS: Вакуумное оборудование установки выключено
	VacuumedUnit:			BOOL; //STAUTS: Установка под вакуумом
	DevacuumedUnit:			BOOL; //STATUS: Установка под атмосферой 
END_STRUCT
END_TYPE

// Structs/Pumping/VacuumProccessWithSHV/VacuumProccessStatus
TYPE VacuumProccessStatus :
UNION
	Status: WORD;
	bStatus: udtVacuumProccessStatusBitMap;
END_UNION
END_TYPE

// Structs/Pumping/VacuumProccessWithSHV/VacuumStage
{attribute 'qualified_only'}
{attribute 'strict'}
TYPE VacuumStage :
(
	WAIT := 0,
	START_UNIT:=20,
	START_UNIT_COMPETE:=30,
	DEVACUUM:=40,
	DEVACUUM_COMPLETE:=50,
	REVACUUM:=60,
	REVACUUM_COMPLETE:=70,
	STOP_UNIT:=80,
	STOP_UNIT_COMPLETE:=90,
	ERROR:=1000
);
END_TYPE

// Structs/RRG/Modbus/udtRRGFlagState1
TYPE udtRRGFlagState1 :
UNION
	bState:WORD;
	Flags: udtRRGFlagState1Flags;
END_UNION
END_TYPE

// Structs/RRG/Modbus/udtRRGFlagState1Flags
TYPE udtRRGFlagState1Flags :
STRUCT
	N_1:			BIT;
	DigitalInput: 	BIT; //0 - Analog Input; 1-Digital Input
	StateBit2:		BIT;
	StateBit3: 		BIT;
	RepareBit: 		BIT; // 0 -Система восстановится в цифровом управлении; 1-Система восстановится в аналоговом управлении
	RRGMode: 		BIT; // 0 - RRG; 1 - RRD
	SetZero: 		BIT; //  1 - set zero
	N_2:			BIT;
	N_3:			BIT;
	N_4:			BIT;
	N_5:			BIT;
	N_6:			BIT;
	N_7:			BIT;
	N_8:			BIT;
	N_9:			BIT;
	N_10:			BIT;
END_STRUCT
END_TYPE

// Structs/RRG/Modbus/udtRRGFlagState2
TYPE udtRRGFlagState2 :
UNION
	bState:WORD;
	Flags: udtRRGFlagState2Flags;
END_UNION
END_TYPE

// Structs/RRG/Modbus/udtRRGFlagState2Flags
TYPE udtRRGFlagState2Flags :
STRUCT
	LowGasFlow: 	BIT; //0 - норма; 1- Недостаточно газа более 20 секунд
	ValveMode: 		BIT;// 0 - затвор в режиме регулирвоания; 1- затвор в двухпозиционном режиме
	RegMode: 		BIT;// 0 - RRG; 1-RDG
	RDGOnly:		BIT;
	RRGOnly:		BIT;
	StateBit5: 		BIT;
	StateBit6:		BIT;
	N_1:			BIT;
	N_3:			BIT;
	N_4:			BIT;
	N_5:			BIT;
	N_6:			BIT;
	N_7:			BIT;
	N_8:			BIT;
	N_9:			BIT;
	N_10:			BIT;
END_STRUCT
END_TYPE

// Structs/RRG/Modbus/udtRRGModbus
TYPE udtRRGModbus :
STRUCT
	Address: 		WORD;
	Number:			WORD;
	FlagState1_Write: 	udtRRGFlagState1;
	FlagState1_Read: 	udtRRGFlagState1;
	FlagState2: 	udtRRGFlagState2;
	GasFlowSPWrite: WORD;
	GasFlowSPRead: WORD;
	GasFlowFB: 		WORD;
	COMPortSpeed:	WORD;
END_STRUCT
END_TYPE

// Structs/TRM151_Control/View/udtTRMChannelView
TYPE udtTRMChannelView :
STRUCT
	
	ChannelNo: INT;		//Номер канала
	xEnablePidRegualtor:	INT; //SETTING: Включить регулятор
	
	



END_STRUCT
END_TYPE

// Structs/TRM151_Control/View/udtTRMInputView
TYPE udtTRMInputView :
STRUCT
	InputNo									:INT;
	SensoreType:							TRMInputSensoreType;
	DigitalFiltertimeConst:					DINT;//Постоянная времени цифрового фильтра
	DigitalFilterConstMin:					DINT:=0;
	DigitalFilterConstMax:					DINT:=1800;
	DigitalFilterLine:						DINT;//полопса цифрового фильтра
	DigitalFilterLineMin:					DINT:=0;
	DigitalFilterLineMax:					DINT:=9999;
	PollingSensoreTime:						REAL;// Период опроса датчика
	PollingSensoreTimeMin:					REAL:=0.3;
	PollingSensoretimeMax:					REAL:=30.0;
	CorrectionOfCharacteresticShift:		DINT;//корекция сдвига харакетристик
	CorrectionOfCharacteristicShiftMin:		DINT:= -999;
	CorrectionOfCharacteristicShiftMax:		DINT:=9999;
	CorrectionOfInclineCharacteristic:		REAL;//Коррекция наклона характеристик от 0,9 до 1,1
	CorrectionOfInclineCharacteristicMin:	REAL:=0.9;
	CorrectionOfInclineCharacterisitcMax:	REAL:=1.1;
	LowEdgeSensoreChange:					DINT;//Нижняя граница изменения активного датчика
	LowEdgeSensoreChangeMin:				DINT:= -999;
	LowEdgeSensoreChangeMax:				DINT:=9999;
	HightEdgeSensoreChange:					DINT;//Верхняя граница измений активного датчика
	HightEdgeSensoreChangeMin:				DINT:=-999;
	HightEdgeSensoreChangeMax:				DINT:=9999;
	(*EVENTS*)
	xSaveEvent:								BOOL;//Сигнал о сохранении
END_STRUCT
END_TYPE

// Structs/TRM151_Control/View/udtTRMOutput
TYPE udtTRMOutput :
STRUCT
	OutpudId:						INT;
	MaxSpeedOutputPowerSpeed:		REAL; //Максимальная скорость изменения выходной мощности
	MaxSpeedOutputPowerSpeedMin:	REAL:=0;
	MaxSpeedOutputPowerSpeedMax:	REAL:=100;
	MaxOutputPower:					REAL; //Максимальная выходная можщность
	MaxOutputPowerMin:				REAL:=-100.0;
	MaxOutputPowerMax:				REAL:=100.0;
	MinOutputPower:					REAL;
	MinOutputPowerMin:				REAL:=-100.0;
	MinOutputPowerMax:				REAL:=100.0;
	(*EVENTS*)
	xSaveEvent:						BOOL;//Событие сохранение значений
END_STRUCT
END_TYPE

// Structs/TRM151_Protocol/Calculator/udtCalculator
TYPE udtCalculator :
STRUCT
	CalculatorID:					INT;//Ииндекс вычислиетля 0,8...56
	CalcFormula:					OwenValue:=(ParameterName:='CAL.t');//Формула вычислителя. 0-повтороитель; 1-Взвешенная сумма; 2-Квадратный корень; 3-Частное; 4-Максимум; 5-Минимум; 6 -Медиана; 7-Среднее арифмитическое; 8 -Вычислитель влажности; 9-ВычислительОтключен
	PsychometricCoeffForWetCalc:	OwenValue:=(ParameterName:='A.ist');//STORED_DOT3 Психометрический коэффийиент для расчета влажности 0,064...0,14 
	TimeConstOfDigitalFilter:		OwenValue:=(ParameterName:='CL.Fd');//постоянная вренмени цифрового фильтра 0...1800
	DigitalFilterLine:				OwenValue:=(ParameterName:='CL.FG');//Полоса цифрового фильтра 0...9999
	DecPointPostion:				OwenValue:=(ParameterName:='dP');//Кол-во знаков после десятичной точки на индикаторе 0...3
	CalcArgumentsCount:				OwenValue:=(ParameterName:='n.in.C');//кол-во аргументов вычислителя
	CalcualtorInput:				ARRAY [0..8] OF udtCalculatorInput;			
END_STRUCT
END_TYPE

// Structs/TRM151_Protocol/Calculator/udtCalculatorInput
TYPE udtCalculatorInput :
STRUCT
	InputID:			INT; //Идентификатор входа
	InputDevice:		OwenValue:=(ParameterName:='t.in.');//Тип аругмента вы числителя 
	InputDeviceNumber:	OwenValue:=(ParameterName:='in.');//Номер (считая с нуля) Входа.
	WeightCoeff:		OwenValue:=(ParameterName:='SCA');//Stored DOT Весовой коэффициент для формулы "Взвешенная сумма"
END_STRUCT
END_TYPE

// Structs/TRM151_Protocol/Calculator/udtCalculators
TYPE udtCalculators :
STRUCT
	ComputerAccess:		OwenValue:=(ParameterName:='A.CAL');//ограничесние досутпа к Вычислителям
	Calculator: ARRAY [0..7] OF udtCalculator;
END_STRUCT
END_TYPE

// Structs/TRM151_Protocol/Inputs/udtInput
TYPE udtInput :
STRUCT
	InputNo:							INT;//Номер входа
	SensoreType:						OwenValue:=(ParameterName:='in-t', 	ValueType:=OWEN_TYPE.INTEGER);//Тип датчика
	DigitalFilterTimeConstant:			OwenValue:=(ParameterName:='in.Fd',	ValueType:=OWEN_TYPE.INTEGER);//Постоянная времени цифрового фильтра.0...1800[c]
	DigitalFilterline:					OwenValue:=(ParameterName:='in.FG', ValueType:=OWEN_TYPE.FLOAT);//STORED_DOT Полоса цифрового фильтра 0...9999
	PollingSensoreTime:					OwenValue:=(ParameterName:='itrL', 	ValueType:=OWEN_TYPE.FLOAT);//STORED_DOT1 Период опроса датчика 0,3...30 секунд
	CorrectionOfShiftCharacteristic: 	OwenValue:=(ParameterName:='in.SH', ValueType:=OWEN_TYPE.FLOAT);//STORED_DOT Коррекция "сдвиг харакетристики" -999...9999
	CorrectionOfInclineCharacterisitc:	OwenValue:=(ParameterName:='in.SL', ValueType:=OWEN_TYPE.FLOAT);//STORED_DOT3 коррекция "Наклона характеристики" 0,9....1,1
	LowEdgeSensoreChange:				OwenValue:=(ParameterName:='Ain.L', ValueType:=OWEN_TYPE.FLOAT);//нНижняя граница изменения активного датчика. -999...9999
	HightEdgeSensoreChange:				OwenValue:=(ParameterName:='Ain.H', ValueType:=OWEN_TYPE.FLOAT);//Верхняя граница изменения активного датчика. -999...9999
	InputGroupAttribute:				OwenValue:=(ParameterName:='dt', 	ValueType:=OWEN_TYPE.INTEGER);//Групповой атрибут входа
END_STRUCT
END_TYPE

// Structs/TRM151_Protocol/Inputs/udtInputs
TYPE udtInputs :
STRUCT
	AccessLimit:							OwenValue:=(ParameterName:='A.Mes', ValueType:=OWEN_TYPE.INTEGER);//Огарнчиение доступа. 0 - только по паролю; 1- чтение без пароля; 2-пароль не нужен
	GroupAttrubuteInputsTree:				OwenValue:=(ParameterName:='O.Mes', ValueType:=OWEN_TYPE.INTEGER);//Групповой аттрибут дерева входы. 1-Не редакируемый, заводской; 2-Редактируемый, Заводской; 3-Не редактируемыый, пользовательский; 4- Редактируемый, Пользоватлеьский
	CorrectionModeFromFreeEndsTemperature: 	OwenValue:=(ParameterName:='Cj-.C', ValueType:=OWEN_TYPE.INTEGER );//режим корреции по температуре свободных концов ТП. 1-Выключено; 2- Включен
	Input: ARRAY [0..1] OF udtInput;
END_STRUCT
END_TYPE

// Structs/TRM151_Protocol/LockAndChangeMode/udtTRMLockAndChangeMode
TYPE udtTRMLockAndChangeMode :
STRUCT
	ManuaControl: OwenValue:=(ParameterName:='bL.rU', ValueType:=OWEN_TYPE.INTEGER);
END_STRUCT
END_TYPE

// Structs/TRM151_Protocol/OperationParameters/udtOperationParameters
TYPE udtOperationParameters :
STRUCT
	PowerFeedback:				ARRAY [0..1] OF udtPowerFeedback;
	RegulatorSetPointfeedback:	ARRAY [0..7] OF udtSetPointFeedback; 	
	ProgramNumberFeedback:	OwenValue:=(ParameterName:='r.PrG', ValueType:=OWEN_TYPE.INTEGER);
	StepNumberFeedback:		OwenValue:=(ParameterName:='r.StP', ValueType:=OWEN_TYPE.INTEGER);
	StatusFeedback:			OwenValue:=(ParameterName:='r.St', ValueType:=OWEN_TYPE.INTEGER);
	StarCommand:			OwenValue:=(ParameterName:='r-S', ValueType:=OWEN_TYPE.INTEGER); //0-Stop: 1-Run: 2-pause
END_STRUCT
END_TYPE

// Structs/TRM151_Protocol/OperationParameters/udtPowerFeedback
TYPE udtPowerFeedback :
STRUCT
	ChannelId:	INT;
	Value:		OwenValue:=(ParameterName:='r.out', ValueType:=OWEN_TYPE.FLOAT);
END_STRUCT
END_TYPE

// Structs/TRM151_Protocol/OperationParameters/udtSetPointFeedback
TYPE udtSetPointFeedback :
STRUCT
	RegulatorId: INT;
	Value: OwenValue:=(ParameterName:='Set.P', ValueType:=OWEN_TYPE.FLOAT);
END_STRUCT
END_TYPE

// Structs/TRM151_Protocol/Program/udtProgram
TYPE udtProgram :
STRUCT
	ProgramNumber: 		INT;//0,10,..,110
	StarProgrammAccept: OwenValue:=(ParameterName:='mPr', ValueType:=OWEN_TYPE.INTEGER);//Разрешение на запуск программы. 1-Разрешить; 2-Запретить
	Steps:				ARRAY[0..9] OF udtStep;
END_STRUCT
END_TYPE

// Structs/TRM151_Protocol/Program/udtProgramOfTechnolog
TYPE udtProgramOfTechnolog :
STRUCT
	AccessAttribute: 	OwenValue:=(ParameterName:='pa.lp', ValueType:=OWEN_TYPE.INTEGER);//Аттрибуты доступа. 1-Только по паролю; 2-чтение без пароля; 3-пароль не нужен
	TreeAtribute:		OwenValue:=(ParameterName:='at.lp', ValueType:=OWEN_TYPE.INTEGER);//Групповой аттрибут дерева программы технолога; 1-Не редактиуермы, заводской; 2-Редактируемый, заводской; 3-Не редактиуремый, пользовательский; 4-редактируемый, пользовательский
	TimeScaleInProgram:	OwenValue:=(ParameterName:='t.scl', ValueType:=OWEN_TYPE.INTEGER);//Масштаб времени в программах. 1-Часы-минуты; 2-минуты-секунды
	StartProgramSource:	OwenValue:=(ParameterName:='Str.s', ValueType:=OWEN_TYPE.INTEGER);//Источник запуска программы. 1- Собственная логика; 2-Сетевая коммандаы
	Programs:			ARRAY[0..11] OF udtProgram;
END_STRUCT
END_TYPE

// Structs/TRM151_Protocol/Program/udtStep
TYPE udtStep :
STRUCT
	StepId:								INT;//Индекс шага
	StepType:							OwenValue:=(ParameterName:='st.ty', ValueType:=OWEN_TYPE.INTEGER);//Тип шага. 1-Обычный шаг; 2-Шаг с переходом; 3-Конец программы
	ProgramNumberToTransition:			OwenValue:=(ParameterName:='nu.Pr', ValueType:=OWEN_TYPE.INTEGER);//Нмоер програмы для перехода
	StepNumberToTransition:				OwenValue:=(ParameterName:='nu.St', ValueType:=OWEN_TYPE.INTEGER);//Номер шага для перехода
	NextStepTransitionLogic:			OwenValue:=(ParameterName:='LG.PS', ValueType:=OWEN_TYPE.INTEGER);//Логика перехода на следующий шаг. 1-По достижению порогового значения; 2-По времени; 3-По пороговому з начению и вреемени; 4-по пороговому значению или времени
	SPTransitionCondition:				OwenValue:=(ParameterName:='Sn.PS', ValueType:=OWEN_TYPE.INTEGER);//Условие при переходе "по пороговому значению". 1-Переход если стило меньше порога; 2-переход если стало больше порога
	ComputeNumberValueSourceToTrasition:OwenValue:=(ParameterName:='in.PS', ValueType:=OWEN_TYPE.INTEGER);//Номер вычислителя-источника величина для перехода. 1-Вычислитель не задан; 2..9 - Вычислитель 1-8
	SPValueToTransition:				OwenValue:=(ParameterName:='SP.PS', ValueType:=OWEN_TYPE.FLOAT);//STRORED_DOT Значение порога для перехода -9999 ... 9999
	StepTime:							OwenValue:=(ParameterName:='t.SP', 	Valuetype:=OWEN_TYPE.OTHER);//CLK_fm Длительность шага
END_STRUCT
END_TYPE

// Structs/TRM151_Protocol/Regulators/udt2PositionRegulator
TYPE udt2PositionRegulator :
STRUCT
	HystTwoPositionReg:					OwenValue:=(ParameterName:='HYS.C', ValueType:=OWEN_TYPE.FLOAT);//Гистрезис двухпозиционного регулятора
	DelayTimeFallEdge:					OwenValue:=(ParameterName:='dL.oF', ValueType:=OWEN_TYPE.OTHER);//CLK_frm Время задержки при переходе с ненулевого уровня
	DelayTimeRiseEdge:					OwenValue:=(ParameterName:='dL.on', ValueType:=OWEN_TYPE.OTHER);//CLK_frm Время задержкм при переходе с нулевого уровня
	MinHoldTimeRiseLevel:				OwenValue:=(ParameterName:='Ht.on', ValueType:=OWEN_TYPE.OTHER);//CLR_frm Минимальное время удержания на ненулевом уровне
	MinHoldTimeFallEdge:				OwenValue:=(ParameterName:='Ht.oF', ValueType:=OWEN_TYPE.OTHER);//CLR_frm Минимальное время удержания на нулевом уровне
END_STRUCT
END_TYPE

// Structs/TRM151_Protocol/Regulators/udtPIDRegulator
TYPE udtPIDRegulator :
STRUCT
	PCoeff:				OwenValue:=(ParameterName:='Pb', 	ValueType:=OWEN_TYPE.FLOAT);//STORED_DOT Полоса пропорциональности
	ICoeff:				OwenValue:=(ParameterName:='ti', 	ValueType:=OWEN_TYPE.OTHER);//CLK_frm Постоянная интегрирования ti
	DIDifF:				OwenValue:=(ParameterName:='td.ti', Valuetype:=OWEN_TYPE.FLOAT);//STORED_DOT3 td/ti-отношение ПД к ПИ
	MaxIntegralLimit:	OwenValue:=(ParameterName:='i.UPr', ValueType:=OWEN_TYPE.FLOAT);//STORED_DOT1 Ограничение макстммума интеграла -100...100
	MinIntegralLimit:	OwenValue:=(ParameterName:='i.min', ValueType:=OWEN_TYPE.FLOAT);//Ограничение минимума интеграла
	NominalPower:		OwenValue:=(ParameterName:='P.nom', ValueType:=OWEN_TYPE.FLOAT);//Номинальная можность -100...100
	CoolerPowerCoeff:	OwenValue:=(ParameterName:='P.CLD', ValueType:=OWEN_TYPE.FLOAT);//Коэффициент мощности холодильника 0,01 ... 10
	AddSpeedChangeSP:	OwenValue:=(ParameterName:='v.SP', ValueType:=OWEN_TYPE.FLOAT);//Доп. скорость изменения уставки
END_STRUCT
END_TYPE

// Structs/TRM151_Protocol/Regulators/udtRegulator
TYPE udtRegulator :
STRUCT
	RegulatorID:						INT;//Индекс регулятора
	Deadband:							OwenValue:=(ParameterName:='db', 	ValueType:=OWEN_TYPE.FLOAT);//STORED_DOT Зона нечувствительности
	RegulatorMode:						OwenValue:=(ParameterName:='rEG.t', ValueType:=OWEN_TYPE.INTEGER);//Режим работы регулятора. 0-двупозиционный; 1-ПИД
	RegulatorConnection:				OwenValue:=(ParameterName:='OD.tP', Valuetype:=OWEN_TYPE.INTEGER);//Что подключено к регулятору. 0-ничего; 1-ПС
	NumberOfConnectionSignalConverter:	OwenValue:=(ParameterName:='r.OD.i',ValueType:=OWEN_TYPE.INTEGER);//Номерп подключения преобразователя сигнала. 0-ПС №1; 1-ПС№2
	LBAControl:							OwenValue:=(ParameterName:='LBA', 	ValueType:=OWEN_TYPE.INTEGER);//Контроль LBA аварии. 0-нет контроля; 1-Есть контроль
	PIDRegulator:						udtPIDRegulator;
	TwoPosRegulator:					udt2PositionRegulator;
END_STRUCT
END_TYPE

// Structs/TRM151_Protocol/Regulators/udtRegulators
TYPE udtRegulators :
STRUCT
	Regulator:	ARRAY[0..7] of udtRegulator;
END_STRUCT
END_TYPE

// Structs/TRM151_Protocol/SetPoint/udtProgramSetPoint
TYPE udtProgramSetPoint :
STRUCT
	Steps: ARRAY [0..9] OF udtStepSetPoint;
END_STRUCT
END_TYPE

// Structs/TRM151_Protocol/SetPoint/udtSetPoints
TYPE udtSetPoints :
STRUCT
	Programs: ARRAY[0..11] OF udtProgramSetPoint;
END_STRUCT
END_TYPE

// Structs/TRM151_Protocol/SetPoint/udtStepSetPoint
TYPE udtStepSetPoint :
STRUCT
	SetpointID:			INT;
	SetPointSpeed:		OwenValue:=(ParameterName:='LF.LU',		ValueType:=OWEN_TYPE.FLOAT); //Скорость выхода на уставку
	SetPointType:		OwenValue:=(ParameterName:='P.-SP', 	ValueType:=OWEN_TYPE.INTEGER); //Тип уставки
	MinSetPoint:		OwenValue:=(ParameterName:='b.CH.L', 	ValueType:=OWEN_TYPE.FLOAT); //STORED_DOT нижнаяя граница задания уставки
	MaxSetPoint:		OwenValue:=(ParameterName:='b.CH.H', 	ValueType:=OWEN_TYPE.FLOAT);//STORED_DOT. Верхняя граница задания уставки
	SetPoint:			OwenValue:=(ParameterName:='SP.LU', 	Valuetype:=OWEN_TYPE.FLOAT);// Значение уставки
END_STRUCT
END_TYPE

// Structs/TRM151_Protocol/SignalConverter/udtSignalConverter
TYPE udtSignalConverter :
STRUCT
	OutputId:						INT;//0,4
	MaxSpeedOutputPowerSpeed:		OwenValue:=(ParameterName:='P.rES', ValueType:=OWEN_TYPE.FLOAT);//STORED_DOT Макусимальная допустимая скорость мзменения выходного сигнала
	MaxOutputPower:					OwenValue:=(ParameterName:='P.Upr', ValueType:=OWEN_TYPE.FLOAT);//Stored_DOT1 Ограничение максимального значения выходного сигнала
	MinOutputPower:					OwenValue:=(ParameterName:='P.min', ValueType:=OWEN_TYPE.FLOAT);//STORED_DOT1 Ограничение минимального значения выходного сигнала
END_STRUCT
END_TYPE

// Structs/TRM151_Protocol/SignalConverter/udtSignalConverters
TYPE udtSignalConverters :
STRUCT
	SignalConverter:	ARRAY[0..1] OF udtSignalConverter;
END_STRUCT
END_TYPE

// Structs/Inficon/InficonType/BitByte/InficonInputStatus
TYPE InficonInputStatus :
UNION
	bValue: ARRAY [0..3] OF BYTE;
	xValue: ARRAY [0..3] OF BitByte ;
END_UNION
END_TYPE

// Structs/Inficon/InficonType/BitByte/InficonLogicstatementStatus
TYPE InficonLogicstatementStatus :
UNION
	bValue:		ARRAY[0..12] OF BYTE;
	xValue:		ARRAY[0..12] OF BitByte;
END_UNION
END_TYPE

// Structs/Inficon/InficonType/BitByte/InficonOutputStatus
TYPE InficonOutputStatus :
UNION
	bValue:	ARRAY[0..4] OF BYTE;
	xValue: ARRAY [0..4] of BitByte;
END_UNION
END_TYPE

// Structs/Inficon/InficonType/Real/REAL3x1
TYPE REAL3x1 :
STRUCT
	rValue:	REAL;
	bValue: ARRAY [0..2] OF BYTE;
END_STRUCT
END_TYPE

// Structs/Inficon/InficonType/Real/REAL41
TYPE REAL41 :
STRUCT
	rValue: REAL;
	bValue: ARRAY[0..3] OF BYTE;
END_STRUCT
END_TYPE

// Structs/Inficon/InficonType/Real/REAL4F31
TYPE REAL4F31 :
STRUCT
	rValue: REAL;
	bValue:	ARRAY[0..3] OF BYTE;
END_STRUCT
END_TYPE

// Structs/Inficon/InficonType/Real/REAL4x2
TYPE REAL4x2 :
STRUCT
	rValue: REAL;
	bValue: ARRAY [0..3] of Byte;
END_STRUCT
END_TYPE

// Structs/Inficon/InficonType/Real/REAL5F32
TYPE REAL5F32 :
STRUCT
	rValue:REAL;
	bValue:ARRAY [0..4] OF BYTE;
END_STRUCT
END_TYPE

// Structs/Inficon/InficonType/Real/REAL5x3
TYPE REAL5x3 :
STRUCT
	rValue: REAL;
	bValue:	ARRAY[0..4] OF BYTE;
END_STRUCT
END_TYPE

// Structs/Inficon/InficonType/Real/REAL6F32
TYPE REAL6F32 :
STRUCT
	rValue: REAL;
	bValue: ARRAY[0..5] OF BYTE;
END_STRUCT
END_TYPE

// Structs/Pumping/VacuumProccessWithSHV/Devacuum/DevacuumUnitStage
{attribute 'qualified_only'}
{attribute 'strict'}
TYPE DevacuumUnitStage :
(
	WAIT := 0,
	CHECK_SYSTEM:=10,
	CLOSE_VALVES:=20,
	WAIT_TIME:=30,
	OPEN_VALVE:=40,
	COMPLETE:=50,
	ERROR:=100
);
END_TYPE

// Structs/Pumping/VacuumProccessWithSHV/Devacuum/udtDevacuumUnitProcessSetting
TYPE udtDevacuumUnitProcessSetting :
STRUCT
	WaitTime:		TIME;//Time for WaitTimer
END_STRUCT
END_TYPE

// Structs/Pumping/VacuumProccessWithSHV/Revacuum/RevacuumStage
{attribute 'qualified_only'}
{attribute 'strict'}
TYPE RevacuumStage :
(
	WAIT := 0,
	CLOSE_BAV3:=10,
	CLOSE_TMP_VALVE:=20,
	WAIT_TIMER:=30,
	OPEN_BAV1SMALL:=40,
	OPEN_BAV1BIG:=50,
	OPEN_BAV2:=60,
	OPEN_SHV:=70,
	COMPLETE:=80,
	ERROR:=1000
);
END_TYPE

// Structs/Pumping/VacuumProccessWithSHV/Revacuum/udtRevacuumProcessSetting
TYPE udtRevacuumProcessSetting :
STRUCT
	WaitTime:		TIME;
END_STRUCT
END_TYPE

// Structs/Pumping/VacuumProccessWithSHV/StartUnitStage/StartUnitStage
{attribute 'qualified_only'}
{attribute 'strict'}
TYPE StartUnitStage :
(
	CLOSE_VALVES := 					0, //Закрытие всех клапанов
	START_FVP:=							10,//Запуск ФВН
	CHECK_FVP:=							20,//Проверка фвн и герметичной линии откачки
	OPEN_FORVACUUM_LINE_VALVE_SMALL:=	30,
	OPEN_FORVACUUM_LINE_VALVE_LARGE:=	40,
	OPEN_TMP_VALVE:=					50,
	START_TMP:=							60,
	OPEN_SHV:=							70,
	CLOSE_FORVACUUM_LINE:=				80,
	COMPLETE:=							90,
	ERROR:=								100,
	WAIT:=								1000
);
END_TYPE

// Structs/Pumping/VacuumProccessWithSHV/StartUnitStage/udtStartUnitProcessSetting
TYPE udtStartUnitProcessSetting :
STRUCT
	FVPCheckTime: TIME; //Время проверки
	FVPCheckPressure: REAL; //Давление в форвакуумной линии для прохождения проверки
	CamPressureForBAV1LargeOpen: REAL; //Давление в камере для открытия клапана форвакуумной линии большого сечения
	StartUntiFinallyPressure:	REAL;
END_STRUCT
END_TYPE

// Structs/Pumping/VacuumProccessWithSHV/StopUnit/StopUnitStage
{attribute 'qualified_only'}
{attribute 'strict'}
TYPE StopUnitStage :
(
	WAIT := 0,
	CLOSE_BAV3_BIG:=10,
	CLOSE_BAV3_SMALL:=20,
	CLOSE_BAV1_BIG:=30,
	CLOSE_BAV1_SMALL:=40,
	TURNOFF_TMP:=50,
	CLOSE_BAV2:=60,
	TURNOFF_FVP:=70,
	COMPLETE:=80,
	ERROR:=1000
);
END_TYPE

// Structs/TRM151_Control/View/Operating/udtTRMOperatingView
TYPE udtTRMOperatingView :
STRUCT
	ProgrammNoSP:				DINT;//SETTING: Старт програаммы
	ProgramStepNoSP:			DINT;//SETTING: Старт программы с нужного шага
	ProgramNoFb:				DINT;
	ProgramStepNoFb:			DINT;
	StartProcessSignal:			TRMStartSignal;//Сигнал Стоп,Старт,Паузаы
	rPowerFeedbackChannel_1:	REAL;
	rPowerFeedbackChannel_2:	REAL;
	rReadfeedbackChannel_1:		REAL;
	rReadfeedbackChannel_2:		REAL;
	rSetpointFeedbackChannel_1:	REAL;
	rSetpointFeedbackChannel_2:	REAL;
	
	
	xSaveSignal:				BOOL;
END_STRUCT
END_TYPE

// Structs/TRM151_Control/View/Regulator/udtTRMPIDRegualtor
TYPE udtTRMPIDRegualtor :
STRUCT
	PCoeff:				REAL;
	ICoeff:				REAL;//Коэффициент в секундах
	DIDiff:				REAL;//Отношение показателя диффиринциального к показателю интегральному
	MaxIntegralLimit:	REAL;//Ограничение максимального показателя игнтегрально сотавляющей
	MaxIntegralLimitMin:REAL:=-100.0;
	MaxIntegralLimitMax:REAL:=100.0;
	MinIntegralLimit:	REAL;//
	MinIntegralLimitMin:REAL:=-100;
	MinIntegralLimitMax:REAL:=100;
	NominalPower: 		REAL:=0.0;
	
	
END_STRUCT
END_TYPE

// Structs/TRM151_Control/View/Regulator/udtTRMRegulatorView
TYPE udtTRMRegulatorView :
STRUCT
	RegulatorID:		INT;
	Deadband:			INT;//Зона нечувствительности
	RegulationMode:		TRMRegulationMode; //Реугуляция 0 - двупозиционный,1 - пид
	PIDRegualtor:		udtTRMPIDRegualtor;
	(*EVENTS*)
	xSaveEvent:			BOOL;//Событие сохранения
END_STRUCT
END_TYPE

// Structs/TRM151_Control/View/SetPoints/udtStepSetPointView
TYPE udtStepSetPointView :
STRUCT
	SetpointSpeed:			REAL;//Скорость выхода уставки 
	SetPointType:			TRMSetpointType;
	MinSetpoint:			REAL;//Минимальная уставка
	MaxSetpoint:			REAL;//максимальная уставка
	Setpoint:				REAL;//Уставка
END_STRUCT
END_TYPE

// Structs/TRM151_Control/View/TechnologProgramm/udtTRMTechnologOperation
(*Структура данных для  обработки действий оператора и основной логики программы 
ДЛя ТРМ. Раздел "ПРОГРАММЫ ТЕХНОЛОГА"*)
TYPE udtTRMTechnologOperation :
STRUCT
	TimeFormat:					TRMTimeFormat; //Масштаб времени в программах
	StartProgramSource:			TRMStartProgramSource; //Источник запуска программы
	StartProgramPermit:			TRMProgramPermit;	//Разрешение на старт программы		
	TechnologOperationProgram:	ARRAY[0..11] OF udtTRMTechnologOperationProgram;
	ProgramNo:					INT;
	StepNo:						INT;
	
	
	
	//---------------------------------Визуальная часть----------------------//
	ViewTechnologOperationProgram:		udtTRMTechnologOperationProgram; //Технология визуализации
	ViewTechnologOperationProgramStep: 	REFERENCE TO udtTRMTechnologOperationProgramStep; //Ссылка на объект шага программы, который берется из объекта ViewTecholoOperationProgram
	ViewStepSetpoint:					REFERENCE TO udtStepSetPointView; //Ссылка на объект уставки в шаге, который берется из объекьта ViewTecholoOperationProgram
	xLoadProgram:						BOOL;
	xSaveProgram:						BOOL;
	xSaveEvent:							BOOL;																			
END_STRUCT
END_TYPE

// Structs/TRM151_Control/View/TechnologProgramm/udtTRMTechnologOperationProgram
(*программа технолога /Программа*)
TYPE udtTRMTechnologOperationProgram :
STRUCT
	
	StartProgramPermit:		TRMProgramPermit;
	Step:					ARRAY [0..9] OF udtTRMTechnologOperationProgramStep;
	StepSetPoint:			ARRAY [0..9] OF udtStepSetPointView;
END_STRUCT
END_TYPE

// Structs/TRM151_Control/View/TechnologProgramm/udtTRMTechnologOperationProgramStep
TYPE udtTRMTechnologOperationProgramStep :
STRUCT
	StepID:						INT;
	StepType:					TRMStepType;
	TransactionProgramNo:		INT;//Номер программы для перехода
	TransactionStepNo:			INT;//Номер шага для прехода
	NextStepTransactionLogic:	TRMNextStepTransactionLogic;
	TransactionConditionValue:	TRMTransactionConditionValue; //условия при переходе "по пороговому значению"
	InputNumberTransactionValue:TRMInputNumberTrancitionValue;// Номер входа, величина с которого должна достичь "значения" SP.PS
	SetPoint:					REAL;
	StepLatency:				REAL;//Длительность шага
	
END_STRUCT
END_TYPE
